// TIA Portal V18 export
ORGANIZATION_BLOCK "Main"   // OB1, LAD, ProgramCycle
TITLE = "Main Program Sweep (Cycle)"
{ S7_Optimized_Access := 'TRUE' }
VERSION : 0.1
// stored: AutoNumber true, IsIECCheckEnabled false, SetENOAutomatically false
   VAR_INPUT
      Initial_Call : Bool;   // Initial call of this OB
      Remanence : Bool;   // =True, if remanent data are available
   END_VAR
BEGIN

REGION Network 1
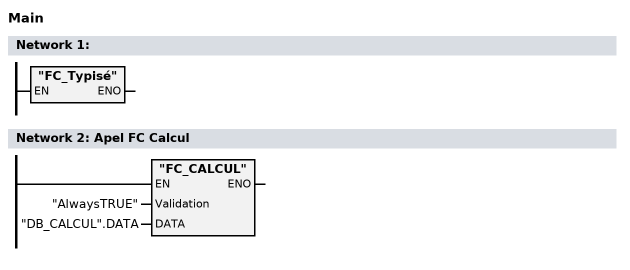
   RUNG wire#powerrail
      "FC_Typisé"()
   END_RUNG
   // the same network as SCL:
   "FC_Typisé"();
END_REGION

REGION Network 2: Apel FC Calcul
   RUNG wire#powerrail
      "FC_CALCUL"(Validation := "AlwaysTRUE", DATA := "DB_CALCUL".DATA)
   END_RUNG
   // the same network as SCL:
   "FC_CALCUL"(Validation := "AlwaysTRUE", DATA := "DB_CALCUL".DATA);
END_REGION
END_ORGANIZATION_BLOCK
